// TIA Portal V16 export
// export: Created 2024-09-05T17:39:19.1237852Z, ExportSetting WithDefaults, DisplayName Totally Integrated Automation Portal, DisplayVersion V16 Update 6, DisplayName TIA Portal Version Control Interface, DisplayVersion V16 Update 2, DisplayName TIA Portal Openness, DisplayVersion V16 Update 6, DisplayName STEP 7 Professional, DisplayVersion V16 Update 6, DisplayName STEP 7 Safety, DisplayVersion V16, DisplayName WinCC Advanced, DisplayVersion V16 Update 6
DATA_BLOCK "AlarmsHandling_DB"   // DB16
VERSION : 0.1
// stored: AutoNumber true, DBAccessibleFromOPCUA true, InstanceOfName AlarmsHandling, InstanceOfType FB
"AlarmsHandling"
   // VAR
   //    IEC_Timer_0_Instance_4 { S7_SetPoint := 'True'} : TON_TIME;
   //    IEC_Timer_0_Instance_5 { S7_SetPoint := 'True'} : TP_TIME;
   //    SetAlarmInstance { S7_SetPoint := 'True'} : Array[0..100] of "SetAlarm_PLC";
   //    AlarmPLCset { S7_SetPoint := 'True'} : Array[0..100] of Program_Alarm;
   // END_VAR
BEGIN
   IEC_Timer_0_Instance_4.PT := T#3S;
   IEC_Timer_0_Instance_4.IN := FALSE;
   IEC_Timer_0_Instance_5.PT := T#0MS;
   IEC_Timer_0_Instance_5.IN := FALSE;
   SetAlarmInstance[0..100].iAlarmCondition := FALSE;
   SetAlarmInstance[0..100].iReset := FALSE;
   SetAlarmInstance[0..14].iTime := T#0MS;
   SetAlarmInstance[15].iTime := T#8S;
   SetAlarmInstance[16..19].iTime := T#5S;
   SetAlarmInstance[20].iTime := T#0MS;
   SetAlarmInstance[21..24].iTime := T#5S;
   SetAlarmInstance[25].iTime := T#0MS;
   SetAlarmInstance[26..28].iTime := T#5S;
   SetAlarmInstance[29..100].iTime := T#0MS;
   SetAlarmInstance[0..100].AlarmToSet := FALSE;
   SetAlarmInstance[0..17].IEC_Timer_0_Instance.PT := T#0MS;
   SetAlarmInstance[18..19].IEC_Timer_0_Instance.PT := T#5S;
   SetAlarmInstance[20..100].IEC_Timer_0_Instance.PT := T#0MS;
   SetAlarmInstance[0..100].IEC_Timer_0_Instance.IN := FALSE;
   SetAlarmInstance[0..100].AlarmToSetWork := FALSE;
END_DATA_BLOCK
